(* CODESYS project e!C_RetainSaveRestore_Test_1.ecp

Project tree, tasks and I/O mapping:
  PFC8202 : 750-8202 PFC200 2ETH RS, WAGO, order no. 0750-8202, version 5.11.1.16
    application Application
      libraries: ; SysPlcCtrl23, 3.5.2.0 (System); VisuDialogs, * (System)
      task PLC_Task (cyclic, interval t#10ms, priority 14) calls PLC_PRG
      task VISU_TASK (cyclic, interval 100 ms, priority 15) calls VisuElems.Visu_Prg
      global variables GPRVL_Test_1
      program PLC_PRG [ST]: RetainTest
      global variables GRVL_Test_1
      visualisation Visu_RetainTest
    DeviceAdapter
    Kbus : Kbus, WAGO, version 1.4.0.2
        unmapped channels: K-BUS diagnostics
    MODBUS
      MODBUS : MODBUS, WAGO, order no. n/a, version 1.1.1.15
    Serial
      COM1 : COM1, WAGO, version 0.0.0.19
  libraries: WagoVisuIcons, 1.0.0.8 (WAGO)
  text list GlobalTextList
*)

// PFC8202/Application/GPRVL_Test_1
VAR_GLOBAL PERSISTENT RETAIN
	wPersistentRetainVar1: WORD := 16#0706;
	wPersistentRetainVar2: WORD := 16#0504;
END_VAR

// PFC8202/Application/GRVL_Test_1
VAR_GLOBAL RETAIN
	wRetainVar1: WORD := 16#0201;
	wRetainVar2: WORD := 16#0403;
END_VAR

// PFC8202/Application/PLC_PRG
PROGRAM PLC_PRG
VAR
	stRetainFileName: STRING := 'RetainFileTest1.bin';
	wRetainCtrlState: WORD;
	xSaveRetain: BOOL;
	xRestoreRetain: BOOL;
	diSaveRetainResult: DINT;
	diRestoreRetainResult: DINT;
	R_TRIG_SaveRetain: R_TRIG;
	R_TRIG_RestoreRetain: R_TRIG;
	TON_RetainCtrlMonitor: TON;
	tSaveRetainMonitor: TIME := T#1S;
END_VAR



RetainTest();

ACTION RetainTest:


wRetainVar1:
wRetainVar2:
wPersistentRetainVar1;
wPersistentRetainVar2;

R_TRIG_SaveRetain(CLK:= xSaveRetain);
R_TRIG_RestoreRetain(CLK:= xRestoreRetain);

CASE wRetainCtrlState OF

	0:(* idle.. *)
		IF (R_TRIG_SaveRetain.Q = TRUE) THEN
			wRetainCtrlState := 10;
		ELSIF (R_TRIG_RestoreRetain.Q = TRUE) THEN
			wRetainCtrlState := 20;
		END_IF

	10:
		diSaveRetainResult := SysSaveRetains(stFileName:= stRetainFileName);
		IF (diSaveRetainResult = 1) THEN
			wRetainCtrlState := 0;
		ELSE
			TON_RetainCtrlMonitor(IN:= TRUE, PT:= tSaveRetainMonitor);
			IF (TON_RetainCtrlMonitor.Q = TRUE) THEN
				TON_RetainCtrlMonitor(IN:= FALSE);
				wRetainCtrlState := 0;
			END_IF
		END_IF

	20:
		diRestoreRetainResult := SysRestoreRetains(stFileName:= stRetainFileName);
		IF (diRestoreRetainResult = 1) THEN
			wRetainCtrlState := 0;
		ELSE
			TON_RetainCtrlMonitor(IN:= TRUE, PT:= tSaveRetainMonitor);
			IF (TON_RetainCtrlMonitor.Q = TRUE) THEN
				TON_RetainCtrlMonitor(IN:= FALSE);
				wRetainCtrlState := 0;
			END_IF
		END_IF

END_CASE
END_ACTION

END_PROGRAM

// PFC8202/Application/Visu_RetainTest
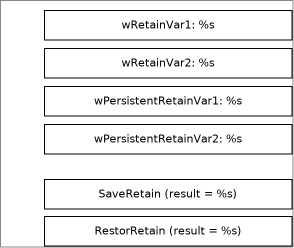
VISUALIZATION Visu_RetainTest  // 294x248
    RoundedRectangle (44,179 248x30), "SaveRetain (result = %s)", text variable: PLC_PRG.diSaveRetainResult
        tap PLC_PRG.xSaveRetain
    RoundedRectangle (44,216 248x30), "RestorRetain (result = %s)", text variable: PLC_PRG.diRestoreRetainResult
        tap PLC_PRG.xRestoreRetain
    RoundedRectangle (44,10 248x30), "wRetainVar1: %s", text variable: wRetainVar1
        OnMouseDown: write the text variable via Default
    RoundedRectangle (44,48 248x30), "wRetainVar2: %s", text variable: wRetainVar2
        OnMouseDown: write the text variable via Default
    RoundedRectangle (44,86 248x30), "wPersistentRetainVar1: %s", text variable: wPersistentRetainVar1
        OnMouseDown: write the text variable via Default
    RoundedRectangle (44,124 248x30), "wPersistentRetainVar2: %s", text variable: wPersistentRetainVar2
        OnMouseDown: write the text variable via Default
END_VISUALIZATION
